INTERFACE ITF_TopElement_HMI

METHOD LinkTopElementData : BOOL
VAR_INPUT
	stData				: REFERENCE TO ST_TopElement_HMI_Link;
END_VAR
END_METHOD

END_INTERFACE

(* stored: Version 1.1.0.1, ProductVersion 3.1.4024.15
   Itf ITF_TopElement_HMI: Id {3b91dccd-4a6c-4fc9-b449-5eb45f3b7186}
   Method LinkTopElementData: Id {80ed8e80-1707-4d86-8843-f28ac024cbfc} *)
